ABB RobotStudio station: Material handiling Assignment.rsstn

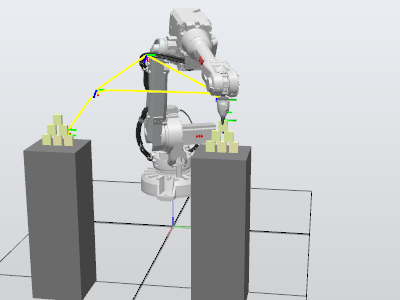
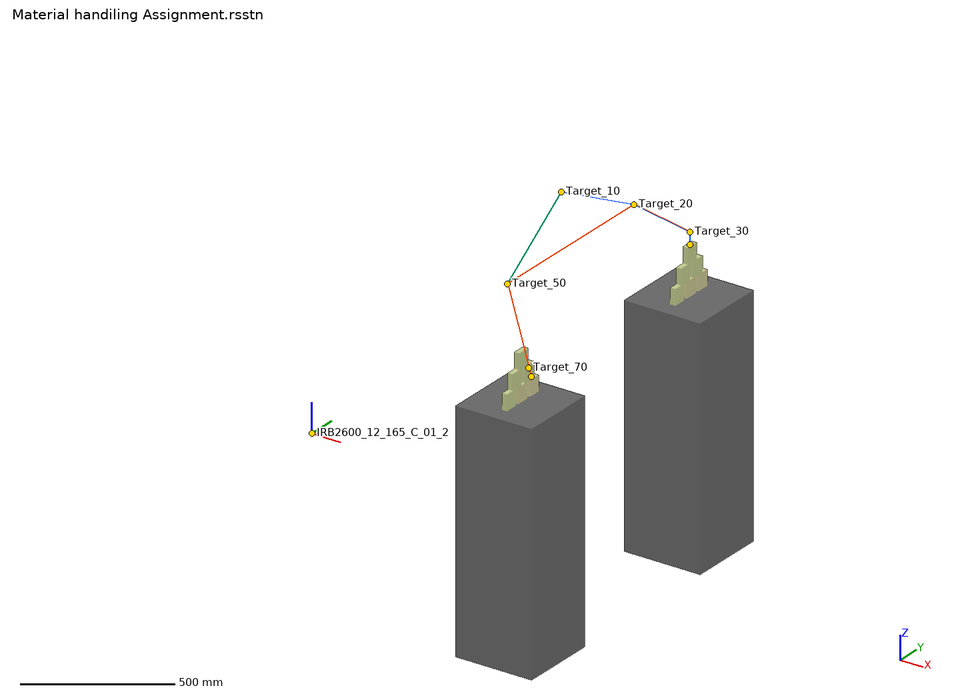
[picture v1: parts stored in the station drawn from their meshes, with robot base, taught points and paths (robot models come from the ABB library and are not in the file)]
Station Station (saved by RobotStudio 22.3.10141.1)
Controller Controller27, task T_ROB1: task frame (RAPID world) sits at (0, 0, 290) mm in the station
Controller Controller27
  mechanical unit ROB_1: IRB2600_12_165_C_01_2, 6 joints, base frame (0, 0, 0) mm
Layout (positions relative to the parent item):
  - Part_1 [part, from Robotics 7020\Cement Base.rslib] at (-450, -450, 0) mm
  - IRB2600_12_165_C_01_2 [mechanism, from %ABB.RobotStudio.Models.IRB2600%\IRB2600_12_165_C_01.rslib] at (0, 0, 290) mm; joint values [0.4247, 0.419, -0.1564, 0.0002, 1.2722, 0.4147] (rad or m)
  - SmartComponent_1 [smart component]
      signals: DI Attach, DO Deatch
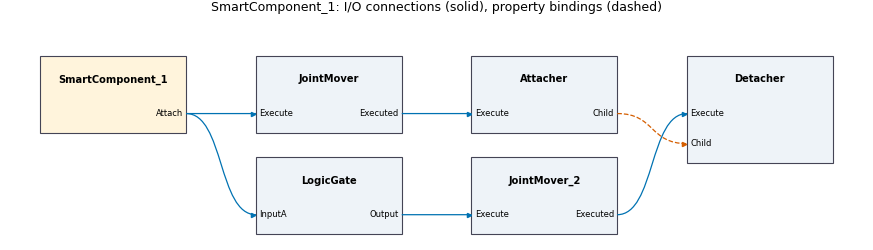
      connections:
        SmartComponent_1.Attach -> JointMover.Execute
        JointMover.Executed -> Attacher.Execute
        SmartComponent_1.Attach -> LogicGate.InputA
        JointMover_2.Executed -> Detacher.Execute
        LogicGate.Output -> JointMover_2.Execute
        Attacher.Child => Detacher.Child
    - Smart_Gripper_Servo_Fingers_2 [mechanism, from Tools\ABB_Smart_Gripper_Servo_Fingers.rslib] at (1125.68, 509.11, 1194.13) mm, rotated rx 179.16 ry 1.88 rz -179.44 deg; joint values [0.025] (rad or m)
    - Detacher [smart component, from Components\Detacher.rslib]
        properties: Child=Part_11; KeepPosition=true
    - Attacher [smart component, from Components\Attacher.rslib]
        properties: Parent=Smart_Gripper_Servo_Fingers_2; Flange=0; Child=Part_11; Mount=false; Offset=[0 0 0]; Orientation=[0 0 0]
    - LogicGate [smart component, from Components\LogicGate.rslib]
        properties: Operator=NOT; Delay=0
    - JointMover [smart component, from Components\JointMover.rslib]
        properties: Mechanism=Smart_Gripper_Servo_Fingers_2; Relative=false; Duration=0; J1=0.02
    - JointMover_2 [smart component, from Components\JointMover.rslib]
        properties: Mechanism=Smart_Gripper_Servo_Fingers_2; Relative=false; Duration=1; J1=0.025
  - Pillerr_1 [part] at (979.41, -592.1, 0) mm, size 300 x 300 x 900 mm
  - Pillerr_2 [part] at (979.41, 355.27, 0) mm, size 300 x 300 x 900 mm
  - Part_3 [part] at (1119.41, 416.03, 900) mm, size 20 x 50 x 60 mm
  - Part_4 [part] at (1119.41, 545.32, 900) mm, size 20 x 50 x 60 mm
  - Part_5 [part] at (1119.41, 480.27, 900) mm, size 20 x 50 x 60 mm
  - Part_8 [part] at (1119.41, 517.74, 960) mm, size 20 x 50 x 60 mm
  - Part_9 [part] at (1119.41, 448.8, 960) mm, size 20 x 50 x 60 mm
  - Part_11 [part] at (1119.41, 485.82, 1020) mm, size 20 x 50 x 60 mm
  - Part_12 [part] at (1119.41, -531.33, 900) mm, size 20 x 50 x 60 mm
  - Part_13 [part] at (1119.41, -402.04, 900) mm, size 20 x 50 x 60 mm
  - Part_14 [part] at (1119.41, -429.63, 960) mm, size 20 x 50 x 60 mm
  - Part_15 [part] at (1119.41, -467.1, 900) mm, size 20 x 50 x 60 mm
  - Part_16 [part] at (1119.41, -498.57, 960) mm, size 20 x 50 x 60 mm
  - Part_17 [part] at (1119.41, -461.54, 1020) mm, size 20 x 50 x 60 mm
  - SmartComponent_2 [smart component]
Attachment: Smart_Gripper_Servo_Fingers_2 is attached to IRB2600_12_165_C_01_2 / Link6
Attachment: SmartComponent_1 is attached to Part_12
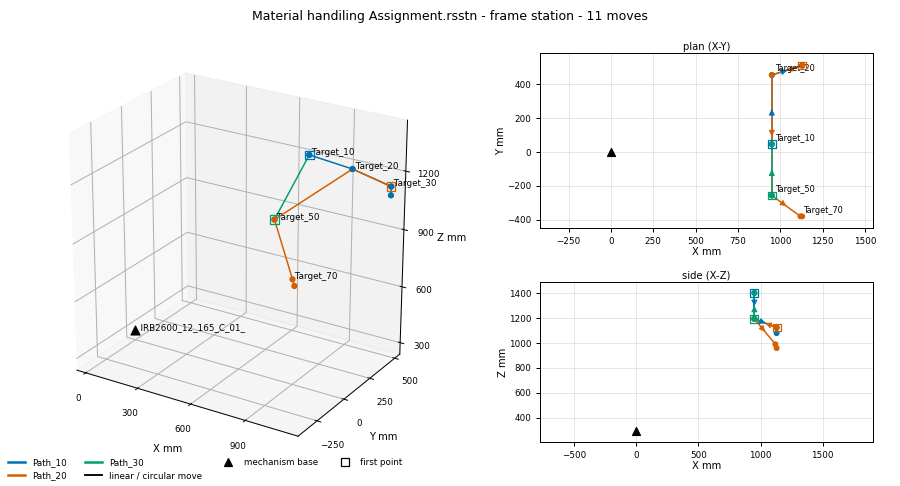
[picture p0: tool path of Material handiling Assignment.rsstn in frame station, 11 of 11 moves have a stored position in this frame; points joined in program order, loops and branches not executed]
Targets, tools, work objects and paths stored in the station, written as RAPID:
! task T_ROB1
MODULE CalibData
  PERS tooldata Servo:=[TRUE,[[0,0,114.2],[1,0,0,0]],[0.215,[8.7,12.3,49.2],[1,0,0,0],0.00021,0.00024,0.00009]];
ENDMODULE

! task T_ROB1
MODULE Module1
  CONST robtarget Target_10:=[[950.282244078,46.028959892,1113.500984511],[0.508914889,0.008286225,0.86065137,0.014703519],[0,-1,0,0],[9E+09,9E+09,9E+09,9E+09,9E+09,9E+09]];
  CONST robtarget Target_20:=[[950.282193968,454.846699407,904.676099003],[0.50891488,0.008286232,0.860651375,0.01470354],[0,-1,0,0],[9E+09,9E+09,9E+09,9E+09,9E+09,9E+09]];
  CONST robtarget Target_30:=[[1129.407035013,510.820899798,835.04964703],[0.01637179,-0.005006568,0.999826109,0.007392595],[0,0,0,0],[9E+09,9E+09,9E+09,9E+09,9E+09,9E+09]];
  CONST robtarget Target_40:=[[1129.407042392,510.820903964,790.00041068],[0.016371803,-0.005006578,0.999826109,0.007392602],[0,0,0,0],[9E+09,9E+09,9E+09,9E+09,9E+09,9E+09]];
  CONST robtarget Target_50:=[[950.282198841,-256.637163219,904.676102457],[0.508914887,0.008286254,0.86065137,0.014703572],[-1,0,-1,0],[9E+09,9E+09,9E+09,9E+09,9E+09,9E+09]];
  CONST robtarget Target_70:=[[1119.407026133,-379.627581067,700.000441632],[0.011969969,-0.014716507,-0.999785908,-0.008263273],[-1,0,-1,0],[9E+09,9E+09,9E+09,9E+09,9E+09,9E+09]];
  CONST robtarget Target_80:=[[1129.407032079,-379.627580245,670.000401039],[0.011970055,-0.01471652,-0.999785907,-0.008263303],[-1,0,-1,0],[9E+09,9E+09,9E+09,9E+09,9E+09,9E+09]];
  PROC Path_10()
    MoveL Target_10,v1000,z100,Servo\WObj:=wobj0;
    MoveL Target_20,v1000,z100,Servo\WObj:=wobj0;
    MoveL Target_30,v1000,z100,Servo\WObj:=wobj0;
    MoveL Target_40,v1000,z100,Servo\WObj:=wobj0;
  ENDPROC
  PROC Path_20()
    MoveL Target_30,v1000,z100,Servo\WObj:=wobj0;
    MoveL Target_20,v1000,z100,Servo\WObj:=wobj0;
    MoveL Target_50,v1000,z100,Servo\WObj:=wobj0;
    MoveL Target_70,v1000,z100,Servo\WObj:=wobj0;
    MoveL Target_80,v1000,z100,Servo\WObj:=wobj0;
  ENDPROC
  PROC Path_30()
    MoveL Target_50,v1000,z100,Servo\WObj:=wobj0;
    MoveL Target_10,v1000,z100,Servo\WObj:=wobj0;
  ENDPROC
  PROC Path_40()
  ENDPROC
ENDMODULE

